// TwinCAT 3 PLC project PLC_B300
// ProgramVersion: 3.1.4024.0
// libraries:
//   Tc2_Standard, * (Beckhoff Automation GmbH)
//   Tc2_System, * (Beckhoff Automation GmbH)
//   Tc3_Module, * (Beckhoff Automation GmbH)
// project tree:
//   DUTs/ stListado_LIQUIDOS.TcDUT
//   / PlcTask.TcTTO
//   POUs/ MAIN.TcPOU

CONFIGURATION PLC_B300
    RESOURCE PLC ON TwinCAT3
        TASK PlcTask(INTERVAL := T#10ms, PRIORITY := 20);
        PROGRAM MAIN WITH PlcTask : MAIN;
    END_RESOURCE
END_CONFIGURATION

// ---- DUTs/stListado_LIQUIDOS.TcDUT
TYPE stListado_LIQUIDOS :
STRUCT
	sProducto:STRING;
	rDensidad:REAL;//g/ml
	iVelAspersor:INT;//velocidad en porcentaje
	bAgitador:BOOL;
	b1000S:BOOL;
	iTempMin:INT;
	iTempMax:INT;
END_STRUCT
END_TYPE

// ---- POUs/MAIN.TcPOU
PROGRAM MAIN
VAR
	bSelecRecetaL01:BOOL;
	bSelecRecetaL02:BOOL;
	bSelecRecetaL03:BOOL;
	bSelecRecetaL04:BOOL;
	bSelecRecetaL05:BOOL;
	bSelecRecetaL06:BOOL;
	bSelecRecetaL07:BOOL;
	bSelecRecetaL08:BOOL;
	bSelecRecetaL09:BOOL;
	bSelecRecetaL10:BOOL;
	bSelecRecetaL11:BOOL;
	bSelecRecetaL12:BOOL;
	bSelecRecetaL13:BOOL;
	bSelecRecetaL14:BOOL;
	bSelecRecetaL15:BOOL;
	bSelecRecetaL16:BOOL;
	bSelecRecetaP1:BOOL;
	bSelecRecetaP2:BOOL;
	bSelecRecetaP3:BOOL;
	bSelecRecetaP4:BOOL;
	iEstadoL01:INT;
	iEstadoL02:INT;
	iEstadoL03:INT;
	iEstadoL04:INT;
	iEstadoL05:INT;
	iEstadoL06:INT;
	iEstadoL07:INT;
	iEstadoL08:INT;
	iEstadoL09:INT;
	iEstadoL10:INT;
	iEstadoL11:INT;
	iEstadoL12:INT;
	iEstadoL13:INT;
	iEstadoL14:INT;
	iEstadoL15:INT;
	iEstadoL16:INT;
	iEstadoP1:INT;
	iEstadoP2:INT;
	iEstadoP3:INT;
	iEstadoP4:INT;
	iRecetaVelMixA1:INT;
	iRecetaVelMixA2:INT;
	iRecetaVelMixA3:INT;
	iRecetaVelAspersor:INT;
	iRecetaTimeHomog:INT;
	iRecetaTimeDescar:INT;
	iRecetaOrden01:INT;
	sRecetaCircuito01:STRING;
	rRecetaDosis01:REAL;
	iRecetaDemora01:INT;
	iRecetaInyec01:INT;
	iRecetaOrden02:INT;
	sRecetaCircuito02:STRING;
	rRecetaDosis02:REAL;
	iRecetaDemora02:INT;
	iRecetaInyec02:INT;
	iRecetaOrden03:INT;
	sRecetaCircuito03:STRING;
	rRecetaDosis03:REAL;
	iRecetaDemora03:INT;
	iRecetaInyec03:INT;
	iRecetaOrden04:INT;
	sRecetaCircuito04:STRING;
	rRecetaDosis04:REAL;
	iRecetaDemora04:INT;
	iRecetaInyec04:INT;
	TablaLiquidos:ARRAY[1..64] OF stListado_LIQUIDOS;
END_VAR

END_PROGRAM
